(* LS Electric XG5000 project: 프로젝트1 *)
(* PLC LSPLC *)

(* Comments on direct variables
%MX0	내부메모리1
%MX1	내부메모리2
*)

PROGRAM NewProgram (* task: 스캔 프로그램 *)
VAR
    result1_1 : BOOL;
    result1_2 : BOOL;
    result1_3 : BOOL;
    result1_4 : BOOL;
    result1_5 : BOOL;
    result1_6 : BOOL;
    result1_7 : BOOL;
    result1_8 : BOOL;
    result2_1 : BOOL;
    result2_2 : BOOL;
    result2_3 : BOOL;
    result2_4 : BOOL;
    result2_5 : BOOL;
    result2_6 : BOOL;
    result2_7 : BOOL;
    result2_8 : BOOL;
    result3_1 : BOOL;
    result3_2 : BOOL;
    result3_3 : BOOL;
    result3_4 : BOOL;
    result3_5 : BOOL;
    result3_6 : BOOL;
    result3_7 : BOOL;
    result3_8 : BOOL;
    result4_1 : BOOL;
    result4_2 : BOOL;
    result4_3 : BOOL;
    result4_4 : BOOL;
    result4_5 : BOOL;
    result4_6 : BOOL;
    result4_7 : BOOL;
    result4_8 : BOOL;
    TON : TON;
    TP : TP;
    경보_냉동_습도램프 AT %QX0.1.24 : BOOL;
    경보_냉동_온도램프 AT %QX0.1.20 : BOOL;
    경보_냉장_습도램프 AT %QX0.1.23 : BOOL;
    경보_냉장_온도램프 AT %QX0.1.19 : BOOL;
    경보_상온_습도램프 AT %QX0.1.21 : BOOL;
    경보_상온_온도램프 AT %QX0.1.17 : BOOL;
    경보_정온_습도램프 AT %QX0.1.22 : BOOL;
    경보_정온_온도램프 AT %QX0.1.18 : BOOL;
    경보냉동상한습도 : WORD := 100;
    경보냉동상한온도 : WORD := -140;
    경보냉동하한습도 : WORD := 10;
    경보냉동하한온도 : WORD := -195;
    경보냉장상한습도 : WORD := 950;
    경보냉장상한온도 : WORD := 110;
    경보냉장하한습도 : WORD := 820;
    경보냉장하한온도 : WORD := 45;
    경보상온상한습도 : WORD := 650;
    경보상온상한온도 : WORD := 270;
    경보상온하한습도 : WORD := 350;
    경보상온하한온도 : WORD := 110;
    경보정온상한습도 : WORD := 580;
    경보정온상한온도 : WORD := -720;
    경보정온하한습도 : WORD := 420;
    경보정온하한온도 : WORD := -870;
    공장가동버튼 AT %IX0.0.0 : BOOL;
    냉동가습기 AT %QX0.1.16 : BOOL;
    냉동가습기수동 AT %IX0.0.16 : BOOL;
    냉동난방기 AT %QX0.1.14 : BOOL;
    냉동난방기수동 AT %IX0.0.14 : BOOL;
    냉동냉방기 AT %QX0.1.13 : BOOL;
    냉동냉방기수동 AT %IX0.0.13 : BOOL;
    냉동상한습도 AT %MW43 : WORD;
    냉동상한온도 AT %MW41 : WORD;
    냉동제습기 AT %QX0.1.15 : BOOL;
    냉동제습기수동 AT %IX0.0.15 : BOOL;
    냉동하한습도 AT %MW42 : WORD;
    냉동하한온도 AT %MW40 : WORD;
    냉동현재습도 AT %MW9 : WORD;
    냉동현재온도 AT %MW5 : WORD;
    냉장가습기 AT %QX0.1.12 : BOOL;
    냉장가습기수동 AT %IX0.0.12 : BOOL;
    냉장난방기 AT %QX0.1.10 : BOOL;
    냉장난방기수동 AT %IX0.0.10 : BOOL;
    냉장냉방기 AT %QX0.1.9 : BOOL;
    냉장냉방기수동 AT %IX0.0.9 : BOOL;
    냉장상한습도 AT %MW33 : WORD;
    냉장상한온도 AT %MW31 : WORD;
    냉장제습기 AT %QX0.1.11 : BOOL;
    냉장제습기수동 AT %IX0.0.11 : BOOL;
    냉장하한습도 AT %MW32 : WORD;
    냉장하한온도 AT %MW30 : WORD;
    냉장현재습도 AT %MW8 : WORD;
    냉장현재온도 AT %MW4 : WORD;
    상온가습기 AT %QX0.1.4 : BOOL;
    상온가습기수동 AT %IX0.0.4 : BOOL;
    상온난방기 AT %QX0.1.2 : BOOL;
    상온난방기수동 AT %IX0.0.2 : BOOL;
    상온냉방기 AT %QX0.1.1 : BOOL;
    상온냉방기수동 AT %IX0.0.1 : BOOL;
    상온상한습도 AT %MW13 : WORD;
    상온상한온도 AT %MW11 : WORD;
    상온제습기 AT %QX0.1.3 : BOOL;
    상온제습기수동 AT %IX0.0.3 : BOOL;
    상온하한습도 AT %MW12 : WORD;
    상온하한온도 AT %MW10 : WORD;
    상온현재습도 AT %MW6 : WORD;
    상온현재온도 AT %MW2 : WORD;
    자동수동전환버튼1 AT %IX0.0.17 : BOOL;
    자동수동전환버튼2 AT %IX0.0.18 : BOOL;
    자동수동전환버튼3 AT %IX0.0.19 : BOOL;
    자동수동전환버튼4 AT %IX0.0.20 : BOOL;
    정온가습기 AT %QX0.1.8 : BOOL;
    정온가습기수동 AT %IX0.0.8 : BOOL;
    정온난방기 AT %QX0.1.6 : BOOL;
    정온난방기수동 AT %IX0.0.6 : BOOL;
    정온냉방기 AT %QX0.1.5 : BOOL;
    정온냉방기수동 AT %IX0.0.5 : BOOL;
    정온상한습도 AT %MW23 : WORD;
    정온상한온도 AT %MW21 : WORD;
    정온제습기 AT %QX0.1.7 : BOOL;
    정온제습기수동 AT %IX0.0.7 : BOOL;
    정온하한습도 AT %MW22 : WORD;
    정온하한온도 AT %MW20 : WORD;
    정온현재습도 AT %MW7 : WORD;
    정온현재온도 AT %MW3 : WORD;
END_VAR

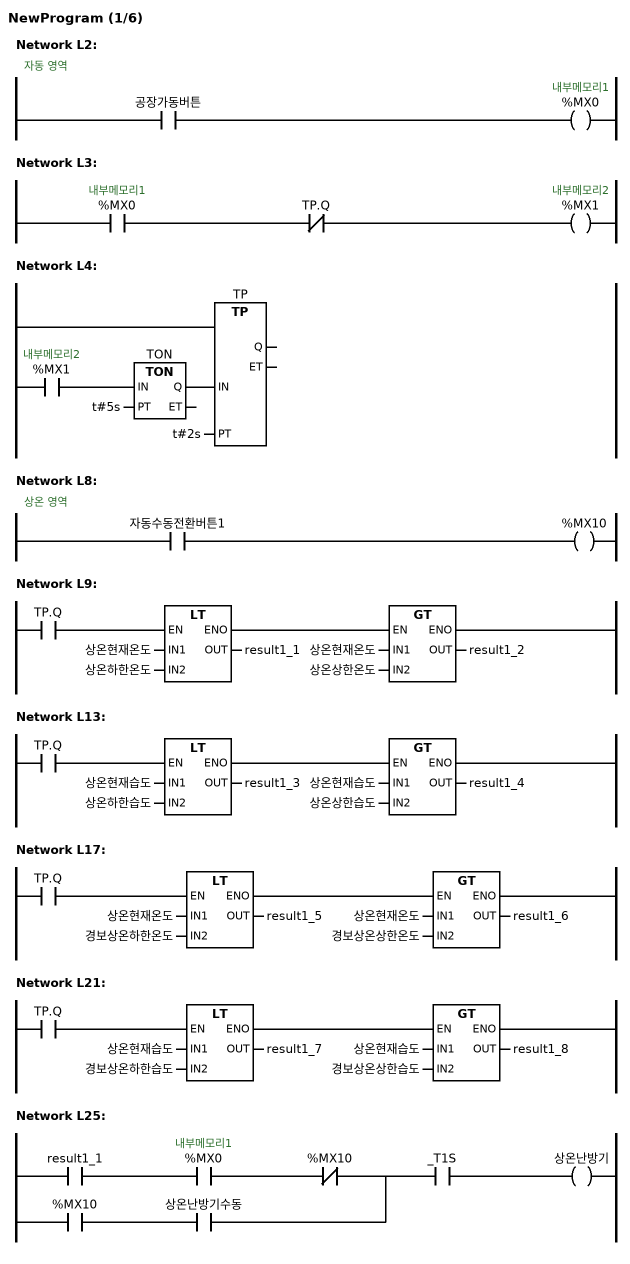
(* 자동 영역 *)
(* Rung L2 *)
%MX0 := 공장가동버튼;
(* Rung L3 *)
%MX1 := %MX0 AND NOT TP.Q;
(* Rung L4 *)
TON(IN := %MX1, PT := t#5s);
TP(IN := TON.Q, PT := t#2s);
(* 상온 영역 *)
(* Rung L8 *)
%MX10 := 자동수동전환버튼1;
(* Rung L9 *)
IF TP.Q THEN
    result1_1 := 상온현재온도 < 상온하한온도;
    result1_2 := 상온현재온도 > 상온상한온도;
END_IF;
(* Rung L13 *)
IF TP.Q THEN
    result1_3 := 상온현재습도 < 상온하한습도;
    result1_4 := 상온현재습도 > 상온상한습도;
END_IF;
(* Rung L17 *)
IF TP.Q THEN
    result1_5 := 상온현재온도 < 경보상온하한온도;
    result1_6 := 상온현재온도 > 경보상온상한온도;
END_IF;
(* Rung L21 *)
IF TP.Q THEN
    result1_7 := 상온현재습도 < 경보상온하한습도;
    result1_8 := 상온현재습도 > 경보상온상한습도;
END_IF;
(* Rung L25 *)
상온난방기 := ((result1_1 AND %MX0 AND NOT %MX10) OR (%MX10 AND 상온난방기수동)) AND _T1S;

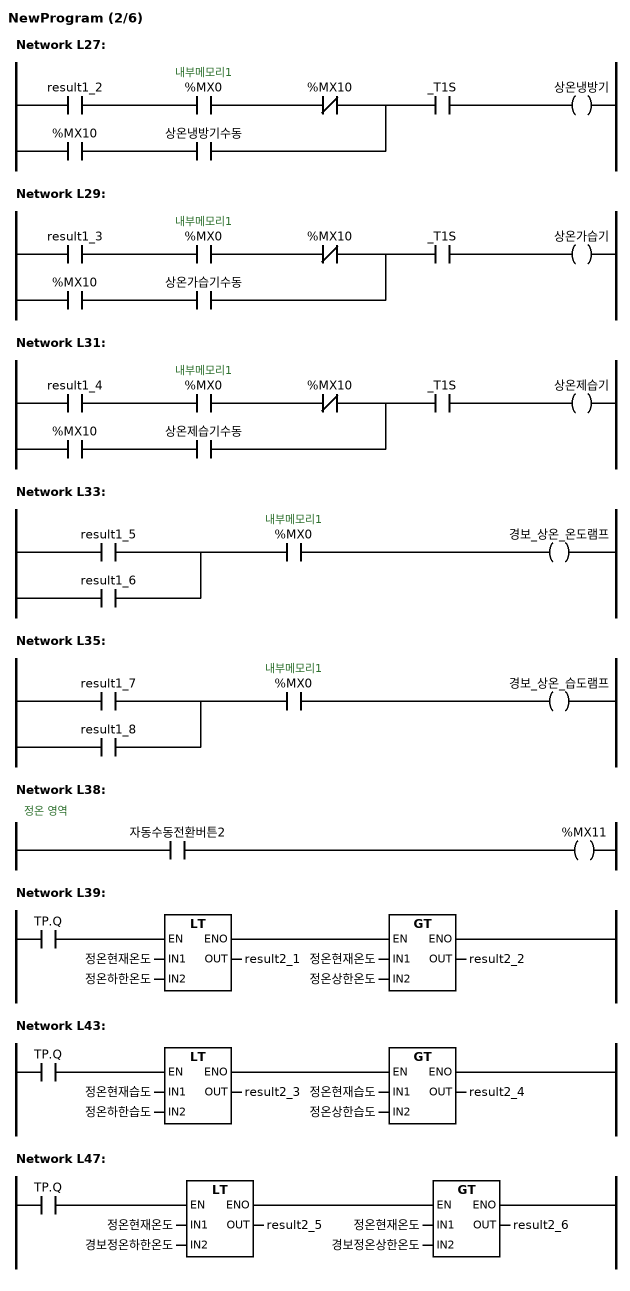
(* Rung L27 *)
상온냉방기 := ((result1_2 AND %MX0 AND NOT %MX10) OR (%MX10 AND 상온냉방기수동)) AND _T1S;
(* Rung L29 *)
상온가습기 := ((result1_3 AND %MX0 AND NOT %MX10) OR (%MX10 AND 상온가습기수동)) AND _T1S;
(* Rung L31 *)
상온제습기 := ((result1_4 AND %MX0 AND NOT %MX10) OR (%MX10 AND 상온제습기수동)) AND _T1S;
(* Rung L33 *)
경보_상온_온도램프 := (result1_5 OR result1_6) AND %MX0;
(* Rung L35 *)
경보_상온_습도램프 := (result1_7 OR result1_8) AND %MX0;
(* 정온 영역 *)
(* Rung L38 *)
%MX11 := 자동수동전환버튼2;
(* Rung L39 *)
IF TP.Q THEN
    result2_1 := 정온현재온도 < 정온하한온도;
    result2_2 := 정온현재온도 > 정온상한온도;
END_IF;
(* Rung L43 *)
IF TP.Q THEN
    result2_3 := 정온현재습도 < 정온하한습도;
    result2_4 := 정온현재습도 > 정온상한습도;
END_IF;
(* Rung L47 *)
IF TP.Q THEN
    result2_5 := 정온현재온도 < 경보정온하한온도;
    result2_6 := 정온현재온도 > 경보정온상한온도;
END_IF;

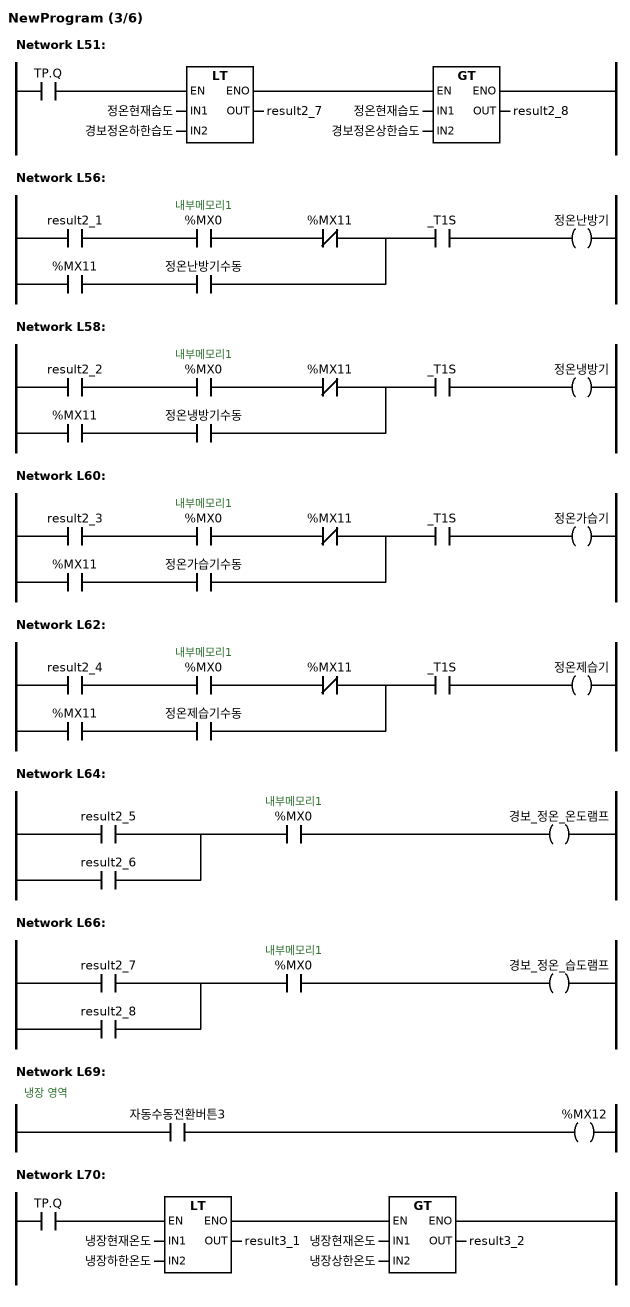
(* Rung L51 *)
IF TP.Q THEN
    result2_7 := 정온현재습도 < 경보정온하한습도;
    result2_8 := 정온현재습도 > 경보정온상한습도;
END_IF;
(* Rung L56 *)
정온난방기 := ((result2_1 AND %MX0 AND NOT %MX11) OR (%MX11 AND 정온난방기수동)) AND _T1S;
(* Rung L58 *)
정온냉방기 := ((result2_2 AND %MX0 AND NOT %MX11) OR (%MX11 AND 정온냉방기수동)) AND _T1S;
(* Rung L60 *)
정온가습기 := ((result2_3 AND %MX0 AND NOT %MX11) OR (%MX11 AND 정온가습기수동)) AND _T1S;
(* Rung L62 *)
정온제습기 := ((result2_4 AND %MX0 AND NOT %MX11) OR (%MX11 AND 정온제습기수동)) AND _T1S;
(* Rung L64 *)
경보_정온_온도램프 := (result2_5 OR result2_6) AND %MX0;
(* Rung L66 *)
경보_정온_습도램프 := (result2_7 OR result2_8) AND %MX0;
(* 냉장 영역 *)
(* Rung L69 *)
%MX12 := 자동수동전환버튼3;
(* Rung L70 *)
IF TP.Q THEN
    result3_1 := 냉장현재온도 < 냉장하한온도;
    result3_2 := 냉장현재온도 > 냉장상한온도;
END_IF;

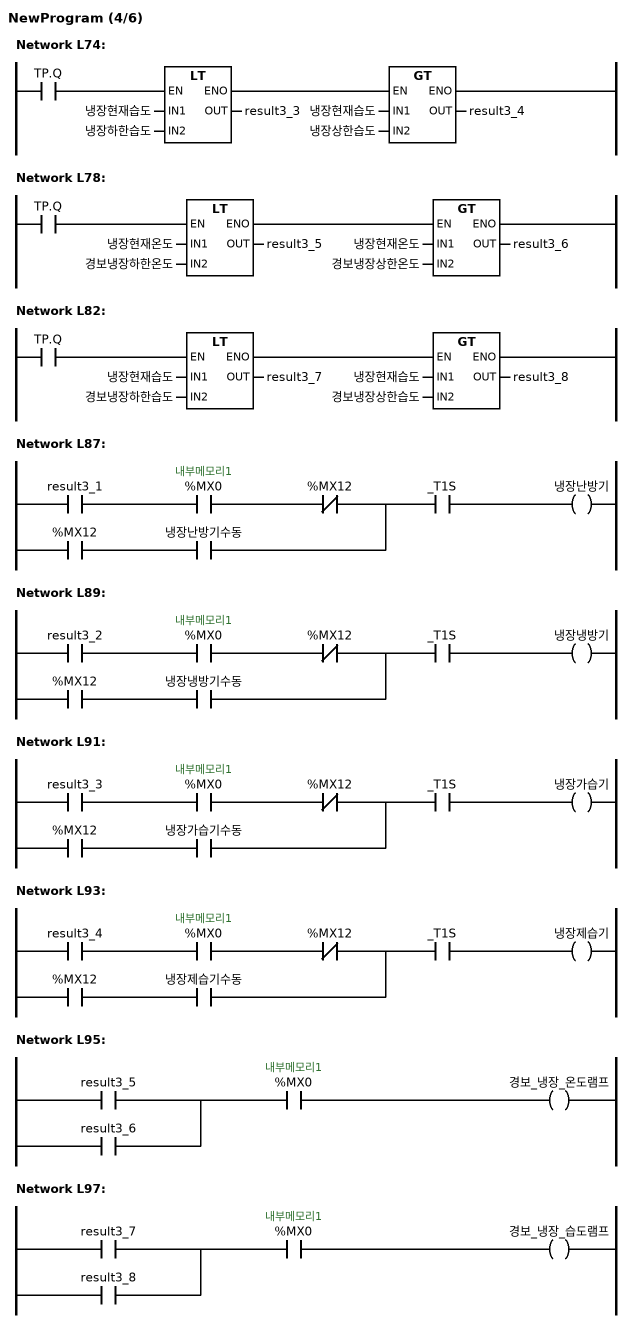
(* Rung L74 *)
IF TP.Q THEN
    result3_3 := 냉장현재습도 < 냉장하한습도;
    result3_4 := 냉장현재습도 > 냉장상한습도;
END_IF;
(* Rung L78 *)
IF TP.Q THEN
    result3_5 := 냉장현재온도 < 경보냉장하한온도;
    result3_6 := 냉장현재온도 > 경보냉장상한온도;
END_IF;
(* Rung L82 *)
IF TP.Q THEN
    result3_7 := 냉장현재습도 < 경보냉장하한습도;
    result3_8 := 냉장현재습도 > 경보냉장상한습도;
END_IF;
(* Rung L87 *)
냉장난방기 := ((result3_1 AND %MX0 AND NOT %MX12) OR (%MX12 AND 냉장난방기수동)) AND _T1S;
(* Rung L89 *)
냉장냉방기 := ((result3_2 AND %MX0 AND NOT %MX12) OR (%MX12 AND 냉장냉방기수동)) AND _T1S;
(* Rung L91 *)
냉장가습기 := ((result3_3 AND %MX0 AND NOT %MX12) OR (%MX12 AND 냉장가습기수동)) AND _T1S;
(* Rung L93 *)
냉장제습기 := ((result3_4 AND %MX0 AND NOT %MX12) OR (%MX12 AND 냉장제습기수동)) AND _T1S;
(* Rung L95 *)
경보_냉장_온도램프 := (result3_5 OR result3_6) AND %MX0;
(* Rung L97 *)
경보_냉장_습도램프 := (result3_7 OR result3_8) AND %MX0;

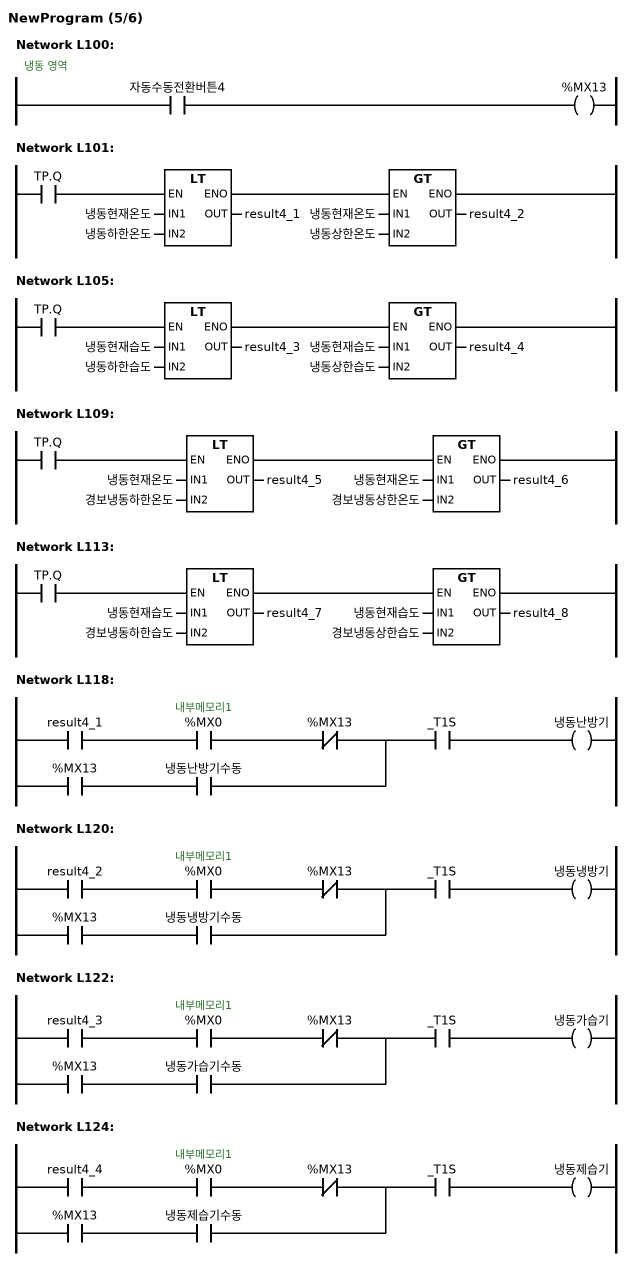
(* 냉동 영역 *)
(* Rung L100 *)
%MX13 := 자동수동전환버튼4;
(* Rung L101 *)
IF TP.Q THEN
    result4_1 := 냉동현재온도 < 냉동하한온도;
    result4_2 := 냉동현재온도 > 냉동상한온도;
END_IF;
(* Rung L105 *)
IF TP.Q THEN
    result4_3 := 냉동현재습도 < 냉동하한습도;
    result4_4 := 냉동현재습도 > 냉동상한습도;
END_IF;
(* Rung L109 *)
IF TP.Q THEN
    result4_5 := 냉동현재온도 < 경보냉동하한온도;
    result4_6 := 냉동현재온도 > 경보냉동상한온도;
END_IF;
(* Rung L113 *)
IF TP.Q THEN
    result4_7 := 냉동현재습도 < 경보냉동하한습도;
    result4_8 := 냉동현재습도 > 경보냉동상한습도;
END_IF;
(* Rung L118 *)
냉동난방기 := ((result4_1 AND %MX0 AND NOT %MX13) OR (%MX13 AND 냉동난방기수동)) AND _T1S;
(* Rung L120 *)
냉동냉방기 := ((result4_2 AND %MX0 AND NOT %MX13) OR (%MX13 AND 냉동냉방기수동)) AND _T1S;
(* Rung L122 *)
냉동가습기 := ((result4_3 AND %MX0 AND NOT %MX13) OR (%MX13 AND 냉동가습기수동)) AND _T1S;
(* Rung L124 *)
냉동제습기 := ((result4_4 AND %MX0 AND NOT %MX13) OR (%MX13 AND 냉동제습기수동)) AND _T1S;

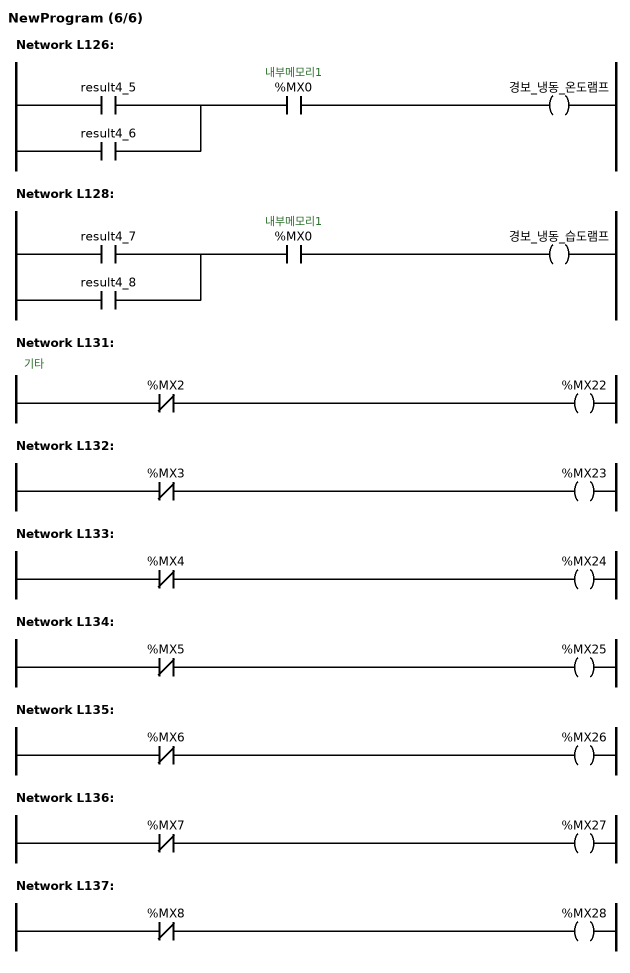
(* Rung L126 *)
경보_냉동_온도램프 := (result4_5 OR result4_6) AND %MX0;
(* Rung L128 *)
경보_냉동_습도램프 := (result4_7 OR result4_8) AND %MX0;
(* 기타 *)
(* Rung L131 *)
%MX22 := NOT %MX2;
(* Rung L132 *)
%MX23 := NOT %MX3;
(* Rung L133 *)
%MX24 := NOT %MX4;
(* Rung L134 *)
%MX25 := NOT %MX5;
(* Rung L135 *)
%MX26 := NOT %MX6;
(* Rung L136 *)
%MX27 := NOT %MX7;
(* Rung L137 *)
%MX28 := NOT %MX8;
END_PROGRAM